(* PLC project canopen_master_slave, beremiz beremiz 1 *)
(* stored: creationDateTime 2008-06-24T18:44:00, contentDescription This example demonstrates PDO communication between a master and a slave CANopen nodes, living in the same PLC. CanFestival CANopen stack's "Virtual" CAN driver is used by default. No real CAN interface and no further configuration are needed, virtual traffic will appear in console. On Linux, SocketCAN driver can be selected instead, implying CAN network configuration such as: ip link set can0 up type can bitrate 125000 ip link set can1 up type can bitrate 125000 Please have a look to https://docs.kernel.org/networking/can.html for more details about Linux SocketCAN support., modificationDateTime 2026-06-01T10:44:41, language en-US *)

PROGRAM test_main_slave
  VAR
    outvar AT %QW0.1.8192.0 : INT;
    invar AT %IW0.1.8193.0 : INT;
  END_VAR

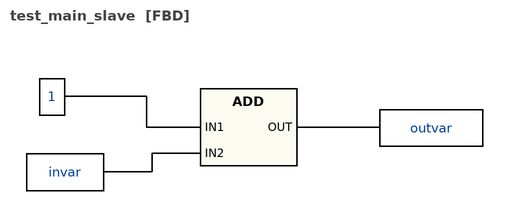
(* FBD diagram, written out as Structured Text *)
outvar := 1 + invar;
END_PROGRAM

PROGRAM test_main_master
  VAR
    PLC_OUT AT %QW0.0.2.8193.0 : INT;
    PLC_IN AT %IW0.0.2.8192.0 : INT;
  END_VAR

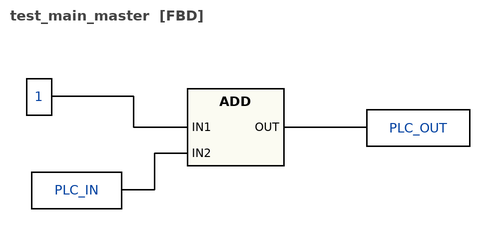
(* FBD diagram, written out as Structured Text *)
PLC_OUT := 1 + PLC_IN;
END_PROGRAM

CONFIGURATION conf
  RESOURCE res ON PLC
    TASK tache(INTERVAL := t#50ms, PRIORITY := 0);
    PROGRAM master WITH tache : test_main_master;
    PROGRAM slave WITH tache : test_main_slave;
  END_RESOURCE
END_CONFIGURATION
